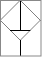
VISUALIZATION VISU_M1Figure_FilterWithDrain  // 42x57
    Polygon (40,20) (20,40) (0,20) (20,0)
    Line (20,40) (20,55)
    Line (10,30) (30,30)
    Line (20,0) (20,30)
END_VISUALIZATION

(* stored: Version 1.1.0.1, ProductVersion 3.1.4019.2
   Visu VISU_M1Figure_FilterWithDrain: Id {fca5ec21-213c-4087-bf16-e2780607163e} *)
